// TIA Portal V19 export
DATA_BLOCK "A0302_Bordatrice"   // DB92
// stored: InstanceOfName A0302_Bordatrice_FB, InstanceOfType FB
"A0302_Bordatrice_FB"
   // VAR_INPUT
   //    AreaInterface : "AreaInterface";
   //    ZSI : "udt_ZoneSafetyInterface";
   //    DSI : "udt_DeviceSafetyInterface";
   //    Drive : "TAx_DriveInterface";
   //    DataIn : Struct
   //       OP : "Ax_PB";
   //       Sens { ExternalAccessible := 'False'; ExternalVisible := 'False'; ExternalWritable := 'False'} : Struct
   //          FTC_Uscita : Bool;
   //       END_STRUCT;
   //       FdBack : Struct
   //          ConnMotori : Bool;
   //          ConnAux : Bool;
   //       END_STRUCT;
   //    END_STRUCT;
   //    CIn { ExternalAccessible := 'False'; ExternalVisible := 'False'; ExternalWritable := 'False'} : Struct
   //       Manager : Struct
   //          Ax : "Positioning_EPOS_Machine_Manager";
   //          Ax_Req : Struct
   //             Pos0 : Bool;
   //             Pos1 : Bool;
   //             Pos2 : Bool;
   //             Pos3 : Bool;
   //          END_STRUCT;
   //       END_STRUCT;
   //       SemiAut_Pb : Bool;
   //       P5 : Struct
   //          Sollevatori : "ValveMachine_COut";
   //          SpintoreLong : "ValveMachine_COut";
   //          Sens : Struct
   //             FTC_Ingombro_A0301 : Bool;
   //          END_STRUCT;
   //       END_STRUCT;
   //       Rulliera : Struct
   //          Ax_1 : "SpeedMachine_COut";
   //          Centratori : "ValveMachine_COut";
   //          Sollevatori : "ValveMachine_COut";
   //          Coda : Struct
   //             Sens : Struct
   //                FTC_Rall : Bool;
   //                FTC_Prox_Ing : Bool;
   //             END_STRUCT;
   //          END_STRUCT;
   //          Centro : Struct
   //             Sens : Struct
   //                FTC_Centrale : Bool;
   //             END_STRUCT;
   //          END_STRUCT;
   //       END_STRUCT;
   //       CarroPareggCoda : Struct
   //          Ax : "Positioning_DOL_Machine_COut";
   //          Bloccaggio : "ValveMachine_COut";
   //          BattutaVerticale : "ValveMachine_COut";
   //          PareggiatoreLongitudinale : "ValveMachine_COut";
   //          Sens : Struct
   //             FTC_Ingombro_In : Bool;
   //             FTC_Ingombro_Out : Bool;
   //             PresenzaMat : Bool;
   //             PosPareggLong : Struct
   //                Value : LReal;
   //                CheckMeasure : Bool;
   //                Standstill : Bool;
   //             END_STRUCT;
   //          END_STRUCT;
   //       END_STRUCT;
   //       CarroPareggTesta : Struct
   //          Ax : "Positioning_DOL_Machine_COut";
   //          Bloccaggio : "ValveMachine_COut";
   //          Centraggio : "ValveMachine_COut";
   //          Sollevatore : "ValveMachine_COut";
   //          Sens : Struct
   //             FTC1_Rall : Bool;
   //             FTC2_Prox_Ls : Bool;
   //             PresenzaMat : Bool;
   //          END_STRUCT;
   //       END_STRUCT;
   //       Attrezzaggio : Struct
   //          CarriParegg : Struct
   //             Ready : Bool;
   //          END_STRUCT;
   //          BordRegFormato : Struct
   //             Ready : Bool;
   //          END_STRUCT;
   //       END_STRUCT;
   //    END_STRUCT;
   //    Config : Struct
   //       Ax : "Positioning_EPOS_Machine_Config_NEW";
   //       Measure : Struct
   //          K1_CarroPost : LReal;
   //          K2_BancoIngresso : LReal;
   //       END_STRUCT;
   //    END_STRUCT;
   //    HWID_TEL111 : HW_SUBMODULE;
   // END_VAR
   // VAR_OUTPUT
   //    MachineInterface { ExternalAccessible := 'False'; ExternalVisible := 'False'; ExternalWritable := 'False'} : "MachineInterface";
   //    DataOut : "Positioning_EPOS_Machine_DataOut";
   //    COut : Struct
   //       Ax : "Positioning_EPOS_Machine_COut";
   //       Ax_VelOveride : Struct
   //          Enable : Bool;
   //          Value : Real;
   //       END_STRUCT;
   //       Sts : Struct
   //          PosTargetEnable : Bool;
   //          PosTarget_Reached : Bool;
   //          In_W_Pos : Bool;
   //          AtRest : Bool;
   //       END_STRUCT;
   //       DataOut : "Positioning_EPOS_Machine_DataOut";
   //    END_STRUCT;
   // END_VAR
   // VAR_IN_OUT
   //    Par : Struct
   //       Ax_Man : "Positioning_EPOS_Machine_Par";
   //       Ax_Aut : "A0301_Mach_Speed_Par";
   //    END_STRUCT;
   //    Pers_Data : Struct
   //       EncoderAbsolute_Preset_OK : Bool;
   //       Persistent_ActualPosition : LReal;
   //    END_STRUCT;
   // END_VAR
   // VAR
   //    Alarm : Struct
   //       Ax { ExternalVisible := 'False'} : "Positioning_EPOS_Machine_Alr";
   //       StopIngombroCarroCoda : Bool;
   //       ConnMotori_FdBack : Bool;
   //       ConnAux_FdBack : Bool;
   //    END_STRUCT;
   //    Warning : Struct
   //       Ax { S7_SetPoint := 'True'} : "Positioning_EPOS_Machine_Wng";
   //       OP_REST_MissingCnd : Bool;
   //       OP_WORK_MissingCnd : Bool;
   //    END_STRUCT;
   //    Ax { S7_SetPoint := 'True'} : "Positioning_EPOS_Machine_FB_NEW";
   //    ValueVelOvr { ExternalAccessible := 'False'; ExternalVisible := 'False'; ExternalWritable := 'False'} : Array[1..10] of Real;
   //    Sts : Struct
   //       ReadyForMove : Bool;
   //       OP_CanMoveFreely : Bool;
   //       OP_MoveToPos_Cnd : Bool;
   //       OP_Bwd_Cnd : Bool;
   //       OP_Fwd_Cnd : Bool;
   //       Pz_UscitaBord : Bool;
   //       StopBordatrice : Bool;
   //       StandbyBordatrice : Bool;
   //    END_STRUCT;
   //    Ctrl : Struct
   //       Bordatrice : Struct
   //          OP_Bwd_Man : Bool;
   //          OP_Fwd_Man : Bool;
   //          OP_Bwd_Aut : Bool;
   //          OP_Fwd_Aut : Bool;
   //          OP_Bwd_Run : Bool;
   //          OP_Fwd_Run : Bool;
   //          OP_MoveToPos : Bool;
   //       END_STRUCT;
   //       Value : Struct
   //          Ax_TargetLongPos { ExternalAccessible := 'False'; ExternalVisible := 'False'; ExternalWritable := 'False'} : LReal;
   //          QuotaInizioUscita : LReal;
   //          QuotaFineUscita : LReal;
   //          PosTarget : LReal;
   //          QuotaRimanenteRullieraCoda : LReal;
   //       END_STRUCT;
   //       PosTargetEnable : Bool;
   //    END_STRUCT;
   //    HMI : Struct
   //       Pos : LReal;
   //    END_STRUCT;
   //    AUX : Struct
   //       Bordatrice : Struct
   //          OP_Bwd_Minus_PB : Bool;
   //          OP_Fwd_Plus_PB : Bool;
   //          OP_MoveToPos_PB { ExternalAccessible := 'False'; ExternalVisible := 'False'; ExternalWritable := 'False'} : Bool;
   //       END_STRUCT;
   //       Measure : Struct
   //          QuotaInizio : Bool;
   //          QuotaFine : Bool;
   //       END_STRUCT;
   //    END_STRUCT;
   //    IEC_FTC_UscitaBordatrice : Struct
   //       TON_Delay : IEC_TIMER;
   //       TOF_Delay { S7_SetPoint := 'True'} : IEC_TIMER;
   //       FTC_On { S7_SetPoint := 'True'} : Bool;
   //    END_STRUCT;
   //    IEC_StandbyBordatrice : IEC_TIMER;
   //    BTrk_Item : Struct
   //       BLean : Real;
   //       O_ID : DInt;
   //    END_STRUCT;
   // END_VAR
BEGIN
END_DATA_BLOCK
